// TIA Portal V20 export
ORGANIZATION_BLOCK "Main"   // OB1, LAD, ProgramCycle
// stored: AutoNumber false
BEGIN

REGION Network 1
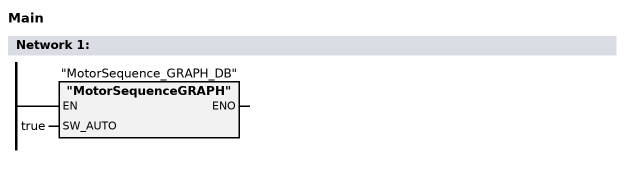
   RUNG wire#powerrail
      "MotorSequence_GRAPH_DB"(SW_AUTO := true)
   END_RUNG
   // the same network as SCL:
   "MotorSequence_GRAPH_DB"(SW_AUTO := true);   // "MotorSequenceGRAPH"
END_REGION
END_ORGANIZATION_BLOCK
